FUNCTION_BLOCK "LGF_ReadPnInterfaceParameter"
TITLE = LGF_ReadPnInterfaceParameter
{ S7_Optimized_Access := 'TRUE' }
AUTHOR : 'Siemens Industry Support'
FAMILY : LGF
NAME : LGF_ReadPnInterfaceParameter
//The function block provides Interface parameter like the IP Address settings, MAC Address and the PN Name.
   VAR_INPUT
      execute : Bool;   // Rising edge starts action once
      hardwareId : HW_ANY;   // Hardware ID of the Interface where the parameter should be read
   END_VAR

   VAR_OUTPUT
      done { ExternalWritable := 'False'} : Bool;   // TRUE: Commanded functionality has been completed successfully
      busy { ExternalWritable := 'False'} : Bool;   // TRUE: FB is not finished, new output values can be expected
      error { ExternalWritable := 'False'} : Bool;   // TRUE: An error occurred during the execution of the FB
      status { ExternalWritable := 'False'} : DWord := #STATUS_NO_CALL;   // 16#0000 - 16#7FFF: Status of the FB, 16#8000 - 16#FFFF: Error identification
      address {InstructionName := 'IP_V4'; LibVersion := '1.0'; ExternalWritable := 'False'} : IP_V4;   // IP Address from interface
      subnetMask {InstructionName := 'IP_V4'; LibVersion := '1.0'; ExternalWritable := 'False'} : IP_V4;   // Subnet mask from interface
      standardGateway {InstructionName := 'IP_V4'; LibVersion := '1.0'; ExternalWritable := 'False'} : IP_V4;   // Standard gateway address from interface
      macAddress { ExternalWritable := 'False'} : Array[0..5] of Byte;   // MAC Address from interface
      pnName { ExternalWritable := 'False'} : String;   // Profinet name from interface
   END_VAR

   VAR
      statExecuteOld { ExternalAccessible := 'False'; ExternalVisible := 'False'; ExternalWritable := 'False'} : Bool;   // Old value of 'execute' input for edge detection
      statDone { ExternalAccessible := 'False'; ExternalVisible := 'False'; ExternalWritable := 'False'} : Bool;   // Static value for output 'done'
      statBusy { ExternalAccessible := 'False'; ExternalVisible := 'False'; ExternalWritable := 'False'} : Bool;   // Static value for output 'busy'
      statError { ExternalAccessible := 'False'; ExternalVisible := 'False'; ExternalWritable := 'False'} : Bool;   // Static value for output 'error'
      statStatus { ExternalAccessible := 'False'; ExternalVisible := 'False'; ExternalWritable := 'False'} : DWord := #STATUS_NO_CALL;   // Static value for output 'status'
      statFBState { ExternalAccessible := 'False'; ExternalVisible := 'False'; ExternalWritable := 'False'} : DInt := #FB_STATE_NO_PROCESSING;   // State in the state machine of the FB
      statHardwareId { ExternalAccessible := 'False'; ExternalVisible := 'False'; ExternalWritable := 'False'} : HW_ANY;   // Hardware ID of the Interface where the parameter should be read
      instRedRec {InstructionName := 'RDREC'; LibVersion := '1.0'; ExternalAccessible := 'False'; ExternalVisible := 'False'; ExternalWritable := 'False'; S7_SetPoint := 'False'} : RDREC;   // Instance for RDREC (Read data record)
      statPdInterfaceData { ExternalAccessible := 'False'; ExternalVisible := 'False'; ExternalWritable := 'False'} : Struct   // Data record for the PN Interface Data
         BlockType { ExternalAccessible := 'False'; ExternalVisible := 'False'; ExternalWritable := 'False'} : UInt;
         BlockLength { ExternalAccessible := 'False'; ExternalVisible := 'False'; ExternalWritable := 'False'} : UInt;
         BlockVersionHigh { ExternalAccessible := 'False'; ExternalVisible := 'False'; ExternalWritable := 'False'} : USInt;
         BlockVersionLow { ExternalAccessible := 'False'; ExternalVisible := 'False'; ExternalWritable := 'False'} : USInt;
         Data { ExternalAccessible := 'False'; ExternalVisible := 'False'; ExternalWritable := 'False'} : Array[0..301] of Byte;
      END_STRUCT;
   END_VAR

   VAR_TEMP
      tempExecute : Bool;   // Temporary value for input 'execute'
      tempIndex : USInt;   // Temporary value for indexing the array
   END_VAR

   VAR CONSTANT
      REC_PDINTERFACE_REAL : DInt := 16#8080;   // Read Record PD Interface
      REC_PDINTERFACE_LENGHT : UInt := 300;   // Read Record PD Interface length
      FB_STATE_NO_PROCESSING : DInt := 0;   // FB state: No processing
      FB_STATE_READ_RECORD : DInt := 1;   // FB state: Reading the data record
      FB_STATE_PROCESS_RECORD : DInt := 2;   // FB state: Process the data record
      STATUS_EXECUTION_FINISHED : Word := 16#0000;   // Execution finished without errors
      STATUS_NO_CALL : Word := 16#7000;   // No job being currently processed
      STATUS_FIRST_CALL : Word := 16#7001;   // First call after incoming new job (rising edge 'execute')
      STATUS_SUBSEQUENT_CALL : Word := 16#7002;   // Subsequent call during active processing without further details
      ERR_UNDEFINED_STATE : Word := 16#9000;   // Error: due to an undefined state in state machine
   END_VAR


BEGIN
	REGION BLOCK INFO HEADER
	  //===============================================================================
	  // SIEMENS / (c)Copyright 2021
	  //-------------------------------------------------------------------------------
	  // Title:            LGF_ReadPnInterfaceParameter
	  // Function:         The function block provides Interface parameter like the IP Address settings, MAC Address and the PN Name.
	  // Library:          LGF
	  // Author:           Siemens Industry Support
	  // Tested with:      CPU 1516-3 PN/DP
	  // Engineering:      TIA Portal V17
	  // Restrictions:     --
	  // Requirements:     S7-1200/1500
	  //-------------------------------------------------------------------------------
	  // Change log table:
	  // Version  | Date       | Expert in charge       | Changes applied
	  //----------|------------|------------------------|------------------------------
	  // 01.00.00 | 2022-12-16 | Siemens Online Support | First released version
	  //===============================================================================
	END_REGION

	REGION DESCRIPTION
	(/*
	The function reads the Interface settings / parameters using the system function `RDREC` (Read data record).

	To read the MAC and IP address of the interface provided via it's hardware ID,
	it is mandatory to read the `PD_INTERFACE_DATA_REAL` data record of any PROFINET compliant interface.

	---

	Note
	:    Upon TIA Portal V17, it’s possible to use as well the system function `CommConfig`, which is in the `Instructions / Communication / Open user communication (Version >= V8.1)` located.
	*/)
	END_REGION DESCRIPTION

	REGION TRIGGERING
	  #tempExecute := #execute; // Work with temporary value / create process image
	  IF (#tempExecute = TRUE) AND (#statExecuteOld = FALSE) // Check if FB is triggered
	    // TODO(optional): delete next line and comment line if FB shall finish current job before new job can be started with rising edge of execute
	    AND (#statStatus = #STATUS_NO_CALL)
	  THEN // First call; initialize FB
	    #statDone := FALSE;
	    #statBusy := TRUE;
	    #statError := FALSE;
	    #statStatus := #STATUS_FIRST_CALL;
	    // State machine - start processing
	    #statFBState := #FB_STATE_READ_RECORD;

	    // Init ariables
	    #statHardwareId := #hardwareId;
	    // PNN Name
	    #pnName := '';
	    // MAC-Address data
	    #macAddress[0] := 16#00;
	    #macAddress[1] := 16#00;
	    #macAddress[2] := 16#00;
	    #macAddress[3] := 16#00;
	    #macAddress[4] := 16#00;
	    #macAddress[5] := 16#00;
	    // IP-Address data
	    #address.ADDR[1] := 16#00;
	    #address.ADDR[2] := 16#00;
	    #address.ADDR[3] := 16#00;
	    #address.ADDR[4] := 16#00;
	    // Subnetmask data
	    #subnetMask.ADDR[1] := 16#00;
	    #subnetMask.ADDR[2] := 16#00;
	    #subnetMask.ADDR[3] := 16#00;
	    #subnetMask.ADDR[4] := 16#00;
	    // Copy Standard Gateway data
	    #standardGateway.ADDR[1] := 16#00;
	    #standardGateway.ADDR[2] := 16#00;
	    #standardGateway.ADDR[3] := 16#00;
	    #standardGateway.ADDR[4] := 16#00;

	    // Initialize functionality: call subsidiary FBs with FALSE
	    #instRedRec(REQ    := FALSE,
	                ID     := #statHardwareId, //Interface to be questioned [HW_ID]
	                INDEX  := #REC_PDINTERFACE_REAL,
	                MLEN   := #REC_PDINTERFACE_LENGHT,
	                RECORD := #statPdInterfaceData);

	  ELSIF (#statStatus = #STATUS_FIRST_CALL) THEN
	    #statStatus := #STATUS_SUBSEQUENT_CALL;
	  END_IF;

	  // Edge detection 'execute' input
	  #statExecuteOld := #tempExecute;
	END_REGION TRIGGERING

	IF (#statStatus = #STATUS_NO_CALL) THEN // Nothing to do -> End here to reduce "system load"
	  RETURN;
	END_IF;

	REGION STATE MACHINE
	  CASE #statFBState OF // State machine of FB
	    #FB_STATE_NO_PROCESSING:
	      REGION No Processing
	        ; // No processing active (Note: this state must always be present and left empty)
	      END_REGION No Processing

	    #FB_STATE_READ_RECORD:
	      REGION Processing Read Record
	        #instRedRec(REQ    := TRUE,
	                    ID     := #statHardwareId, //Interface to be questioned [HW_ID]
	                    INDEX  := #REC_PDINTERFACE_REAL,
	                    MLEN   := #REC_PDINTERFACE_LENGHT,
	                    RECORD := #statPdInterfaceData);

	        IF (#instRedRec.VALID = TRUE) THEN
	          #statFBState := #FB_STATE_PROCESS_RECORD;

	        ELSIF (#instRedRec.ERROR = TRUE) THEN // Error occurred in subsidiary FB
	          #statStatus := #instRedRec.STATUS; // Set status of read record
	        END_IF;
	      END_REGION Processing Read Record

	    #FB_STATE_PROCESS_RECORD:
	      REGION Processing Process the DataRecord
	        // Get PN-interface Name. String starts at an odd address within the array
	        Chars_TO_Strg(Chars  := #statPdInterfaceData.Data,
	                      pChars := 1,
	                      Cnt    := BYTE_TO_UINT(#statPdInterfaceData.Data[0]),
	                      Strg   => #pnName);

	        // Calculate start address of IP-address data. Blockdata is padded to make it Unsigned32 aligned!
	        // When reading is valid, then calculate the offset of the MAC address inside the array
	        #tempIndex := BYTE_TO_USINT(#statPdInterfaceData.Data[0]) + (4 - ((BYTE_TO_USINT(#statPdInterfaceData.Data[0]) + 2) MOD 4));

	        // Copy MAC-Address data
	        #macAddress[0] := #statPdInterfaceData.Data[#tempIndex + 0];
	        #macAddress[1] := #statPdInterfaceData.Data[#tempIndex + 1];
	        #macAddress[2] := #statPdInterfaceData.Data[#tempIndex + 2];
	        #macAddress[3] := #statPdInterfaceData.Data[#tempIndex + 3];
	        #macAddress[4] := #statPdInterfaceData.Data[#tempIndex + 4];
	        #macAddress[5] := #statPdInterfaceData.Data[#tempIndex + 5];

	        // Copy IP-Address data
	        #address.ADDR[1] := #statPdInterfaceData.Data[#tempIndex + 8 + 0];
	        #address.ADDR[2] := #statPdInterfaceData.Data[#tempIndex + 8 + 1];
	        #address.ADDR[3] := #statPdInterfaceData.Data[#tempIndex + 8 + 2];
	        #address.ADDR[4] := #statPdInterfaceData.Data[#tempIndex + 8 + 3];

	        // Copy Subnetmask data
	        #subnetMask.ADDR[1] := #statPdInterfaceData.Data[#tempIndex + 12 + 0];
	        #subnetMask.ADDR[2] := #statPdInterfaceData.Data[#tempIndex + 12 + 1];
	        #subnetMask.ADDR[3] := #statPdInterfaceData.Data[#tempIndex + 12 + 2];
	        #subnetMask.ADDR[4] := #statPdInterfaceData.Data[#tempIndex + 12 + 3];

	        // Copy Standard Gateway data
	        #standardGateway.ADDR[1] := #statPdInterfaceData.Data[#tempIndex + 16 + 0];
	        #standardGateway.ADDR[2] := #statPdInterfaceData.Data[#tempIndex + 16 + 1];
	        #standardGateway.ADDR[3] := #statPdInterfaceData.Data[#tempIndex + 16 + 2];
	        #standardGateway.ADDR[4] := #statPdInterfaceData.Data[#tempIndex + 16 + 3];

	        // Reset Read record
	        #instRedRec(REQ    := FALSE,
	                    ID     := #statHardwareId, //Interface to be questioned [HW_ID]
	                    INDEX  := #REC_PDINTERFACE_REAL,
	                    MLEN   := #REC_PDINTERFACE_LENGHT,
	                    RECORD := #statPdInterfaceData);

	        #statStatus := #STATUS_EXECUTION_FINISHED;
	      END_REGION Processing Process the DataRecord

	    ELSE // Undefined state in state machine reached
	      REGION Undefined state
	        #statStatus := #ERR_UNDEFINED_STATE;
	      END_REGION Undefined state
	  END_CASE;
	END_REGION STATE MACHINE

	REGION OUTPUTS
	  // Write outputs
	  IF (#statStatus = #STATUS_EXECUTION_FINISHED) AND (#statDone = FALSE) THEN // Execution finished without errors
	    REGION Execution finished
	      #statDone := TRUE;
	      #statBusy := FALSE;
	      #statError := FALSE;
	      // execution aborted --> set state no processing
	      #statFBState := #FB_STATE_NO_PROCESSING;
	    END_REGION Execution finished

	  ELSIF (#statStatus.%X15 = TRUE) AND (#statError = FALSE) THEN // Error occurred (#statStatus is 16#8000 to 16#FFFF)
	    REGION Error occured
	      #statDone := FALSE;
	      #statBusy := FALSE;
	      #statError := TRUE;
	      // execution aborted --> set state no processing
	      #statFBState := #FB_STATE_NO_PROCESSING;
	    END_REGION Error occured

	  ELSIF (#tempExecute = FALSE) AND ((#statDone = TRUE) OR (#statError = TRUE)) THEN // Reset outputs
	    REGION Execute reseted
	      #statDone := FALSE;
	      #statBusy := FALSE;
	      #statError := FALSE;
	      #statStatus := #STATUS_NO_CALL;
	    END_REGION Execute reseted
	  END_IF;

	  REGION Write static values to outputs
	    #done := #statDone;
	    #busy := #statBusy;
	    #error := #statError;
	    #status := #statStatus;
	    // if ENO mechanism is not used / not wanted replace the following line by --> ENO := TRUE;
	    ENO := NOT #statError;
	  END_REGION Write static values to outputs
	END_REGION OUTPUTS

END_FUNCTION_BLOCK

